Universal Robots PolyScope program: forcetestwithwaypoint.urp

Program forcetestwithwaypoint (installation=default_4 directory=/programs/usbdisk/new folder_1 createdIn=5.18.0 lastSavedIn=5.18.0 robotSerialNumber=20245388888)
Calibrated DH parameters: a=[0, -0.24355, -0.2132, 0, 0, 0]; d=[0.15185, 0, 0, 0.13105, 0.08535, 0.0921]; alpha=[1.570796, 0, 0, 1.570796, -1.570796, 0]; deltaTheta=[0, 0, 0, 0, 0, 0]
InitVariablesNode
Robot Program (runOnlyOnce=false)
  Force Simple feature=Joint_6_name; selection=[0, 0, 1, 0, 0, 0]; wrench=[0, 0, 5, 0, 0, 0]; limitsForce=[0.15, 0.15, 0.15, 1.047198, 1.047198, 1.047198]; limitsMotion=[0.1, 0.1, 0.1, 0.349066, 0.349066, 0.349066]
    MoveJ speed 60 deg/s, acceleration 80 deg/s^2 (useActiveTCP=true optimoveEnabled=true optiMovePercentage=30) feature=Base
      Waypoint Waypoint_2: TCP in base x=217.156 y=-311.118 z=493.453 mm, rx=-0.9407 ry=1.6463 rz=-1.7185 rad; joints [-34.418, -169.357, 73.18, -84.252, 88.219, -5.67] deg
  MoveJ speed 60 deg/s, acceleration 80 deg/s^2 (useActiveTCP=true optimoveEnabled=true optiMovePercentage=30) feature=Base
    Waypoint Waypoint_1: TCP in base x=85.473 y=-225.982 z=467.073 mm, rx=-0.836 ry=1.5607 rz=-1.8331 rad; joints [-34.447, -169.356, 114.335, -118.232, 85.666, -5.674] deg
